METHOD exe : BOOL
VAR_INPUT
	emergency		:BOOL;		//signal of All_Block and Safety conditions
END_VAR
VAR_IN_OUT
	CMD				:udtCMD;	//standart command word
END_VAR
// Device mode determination
	IF NOT emergency THEN
		//Normal mode
		IF NOT CMD.force THEN
			//No technological lock
			IF NOT CMD.lock AND NOT CMD.alarm AND NOT CMD.service THEN
				//No manual mode
				IF NOT CMD.manual THEN
					CMD.startM := CMD.startA;
				END_IF;
			ELSE
				//Technological lock or device alarm
				CMD.startM := FALSE;
			END_IF;
		END_IF;
	ELSE
		//emergency stop
		CMD.startM := FALSE;
	END_IF;
END_METHOD

METHOD inc : INT
VAR_INPUT
	value			:INT;
	maxValue		:INT;
END_VAR
VAR_IN_OUT
	rotate			:BOOL;
END_VAR
IF rotate THEN
	inc := value + 1;
	IF inc > maxValue THEN
		inc := 0;
	END_IF
	rotate := FALSE;
ELSE
	inc := value;
END_IF
END_METHOD

METHOD blink : BOOL
VAR_INPUT
	req				:BOOL;
	clockOn			:timerRtc;
	clockOff		:timerRtc;
	spOn			:REAL;
	spOff			:REAL;
END_VAR
//blink method
IF req THEN
	//work time
	IF NOT clockOn.cmd.Q AND NOT clockOff.cmd.Q THEN
		blink := TRUE;
		clockOn.cmd.start := TRUE;
	END_IF
	//wait time
	IF clockOn.cmd.Q AND NOT clockOff.cmd.Q THEN
		blink := FALSE;
		clockOff.cmd.start := TRUE;
	END_IF
	//restart time
	IF clockOn.cmd.Q AND clockOff.cmd.Q THEN
		clockOn.cmd.start := FALSE;
		clockOFF.cmd.start := FALSE;
	END_IF
ELSE
	clockOn.cmd.start := FALSE;
	clockOFF.cmd.start := FALSE;
	blink := FALSE;
END_IF

clockOn.sp := spOn;
clockOff.sp := spOff;
sys.timer.rtc(clockOn);
sys.timer.rtc(clockOff);
END_METHOD

METHOD switch : BOOL
VAR_INPUT
	on				:BOOL;
	off				:BOOL;
END_VAR
IF NOT off AND on THEN
	switch := TRUE;
END_IF

IF off THEN
	switch := FALSE;
END_IF
END_METHOD

END_FUNCTION_BLOCK

// System/Library Methods/DrvTimer
FUNCTION_BLOCK DrvTimer
VAR_INPUT
END_VAR
VAR_OUTPUT
END_VAR
VAR
END_VAR

METHOD sec : BOOL
VAR_IN_OUT
	T			:timerSec;		//configuration and command struct for timer of seconds
END_VAR
// Timer with a multiplicity of 1 second
	IF T.CMD.start AND NOT T.CMD.reset THEN
		// Turn on
		IF T.ap < T.sp THEN
			IF NOT T.CMD.pause AND sys.pulse1s THEN
				T.ap := T.ap + 1;
			END_IF;
			T.CMD.Q := FALSE;
		ELSE
			// SP is achieved
			T.CMD.Q := TRUE;
		END_IF;
	ELSE
		// Turn off and reset
		T.ap := 0;
		T.CMD.Q := FALSE;
		T.CMD.reset := FALSE;
	END_IF;
END_METHOD

METHOD cnt : BOOL
VAR_INPUT
	signal 			:BOOL;			//signal from sensor or logical condition
END_VAR
VAR_IN_OUT
	T				:timerCnt;		//configuration and command struct for counter
END_VAR
// Front signal control
	T.PT (CLK := signal);
	
// Timer or counter with free multiplicity 
	IF T.CMD.start AND NOT T.CMD.reset THEN
		// Turn on
		IF NOT T.CMD.pause THEN
			IF T.PT.Q THEN
				T.ap := T.ap + T.one;
			END_IF;
		END_IF;
		//SP control
		IF T.ap < T.sp THEN
			// SP not achieved
			T.CMD.Q := FALSE;
		ELSE
			// SP is achieved
			T.CMD.Q := TRUE;
		END_IF;
	ELSE
		// Turn off and reset
		T.ap := 0.0;
		T.CMD.Q := FALSE;
		T.CMD.reset := FALSE;
	END_IF;

// Progress control
	IF T.sp > 0 AND T.CMD.start THEN
		IF T.ap <= T.sp THEN
			T.percent := (T.ap / T.sp) * 100.0;
		ELSE
			T.percent := 100;
		END_IF
	ELSE
		T.percent := 0.0;
	END_IF;
END_METHOD

METHOD rtc : BOOL
VAR_IN_OUT
	T			:timerRtc;			//configuration and command struct for timer of milliseconds
END_VAR
// Timer with a multiplicity of 1 second
		
	//time counting
	IF T.CMD.start AND NOT T.CMD.reset THEN
		// Turn on
			IF T.RTC = 0 THEN
				T.RTC := sys.upTimeMs;
			END_IF
		//delta calculate
			IF NOT T.CMD.Q THEN
				T.delta := sys.upTimeMs - T.RTC;
			END_IF;
		//delta control
		IF T.ap < T.sp THEN
			T.CMD.Q := FALSE;
		ELSE
			T.CMD.Q := TRUE;
		END_IF;
	ELSE
		// Turn off and reset
		T.ap := 0;
		T.RTC := 0;
		T.delta := 0;
		T.CMD.Q := FALSE;
		T.CMD.reset := FALSE;
	END_IF;
	
	//convert data
		T.ap := UDINT_TO_REAL(T.delta) / 1000;
	
	//calculate time
		IF T.sp > 0 AND T.CMD.start THEN
			T.percent := (T.ap / T.sp) * 100.0;
		ELSE
			T.percent := 0;
		END_IF;
END_METHOD

END_FUNCTION_BLOCK

// Drivers/Devices/03. Analog Input/DrvAI_MV210
FUNCTION_BLOCK DrvAI_MV210
VAR_INPUT
	signal			:udtAI_MV210_101;//Analog input signal from PLC
END_VAR	
VAR_IN_OUT
	CMD				:udtCMD;		//Non-retain structure with command word
	cfg				:cfgAI;			//Retain structure with settings
END_VAR
VAR_OUTPUT
	state			:stateAI_MV210;	//Non-retain structure with states information
	netData			:udtNetDataAnalog;	//Data for network communication via ModBus TCP/RTU
	result			:REAL;			//signal from sensor
END_VAR
VAR
	value			:REAL;			//tmp value for calculating 
	buffer			:REAL;			//tnp value for slow mode
	emergency		:BOOL;			//emergency signal
	cnt				:INT;			//internal counter
	PT				:ARRAY [0..1] OF R_TRIG;
	NT				:ARRAY [0..1] OF F_TRIG;
	clock			:ARRAY [0..3] OF timerRtc;
	Filter			:subFilter;
END_VAR

//ANALOG INPUT
//control of typical analog sensors
// - pressure
// - level
// - flowmeter
// - etc

s00_globalCommands();
IF NOT cfg.cfg.useCompact THEN
	//s01_externalCommand();
	s02_workMode();
	s03_filter();
	s04_alarmsRaw();
END_IF
s05_exe();
//s06_delays();
//s07_turnON();
//s08_turnOFF();
s09_options();
s10_alarms();
s11_reset();
s12_state();
//s13_commands();
//s14_opTime();
s15_globalData();
s16_timers();
s17_hmi();
s18_netData();
//s19_reserv();
//s20_test();

ACTION s07_turnON:

END_ACTION

ACTION s17_hmi:
//hmi data
	//input scaling
		state.signal := sys.base.scale(
			value := signal.signal,
			inputType := cfg.inputType,
			range := cfg.range);
	//rotate input type
		cfg.inputType := sys.base.inc(
			rotate := cmd.test,
			value := cfg.inputType,
			maxValue := sys.aiMaxValueType);
	//rotate value type
		cfg.valueType := sys.base.inc(
			rotate := cmd.lowSpeed,
			value := cfg.valueType,
			maxValue := sys.aiMaxValueValue);
	//rotate filter type
		cfg.filterType := sys.base.inc(
			rotate := cmd.local,
			value := cfg.filterType,
			maxValue := sys.aiMaxValueFilter);
END_ACTION

ACTION s04_alarmsRaw:
//alarms raw
	
	//SC control
	IF cfg.cfg.useSC AND CMD.startA  THEN
		CASE cfg.inputType OF 
			0: 	//0..20 mA
				state.alarm.almSC := sys.base.almS(
					signal := state.signal > 21.0,
					reset := cmd.reset);
			1: 	//4..20 mA
				state.alarm.almSC := sys.base.almS(
					signal := state.signal > 21.0,
					reset := cmd.reset);
				state.alarm.almNC := sys.base.almS(							//NC control only for 4..20 mA
					signal := state.signal < 2.5,
					reset := cmd.reset);
			2: 	//0..10 V
				state.alarm.almSC := sys.base.almS(
					signal := state.signal > 10.5,
					reset := cmd.reset);
			3: 	//-150..+150 C
				state.alarm.almSC := sys.base.almS(
					signal := state.signal > 155.0,
					reset := cmd.reset);
			4: 	//-150..+250 C
				state.alarm.almSC := sys.base.almS(
					signal := state.signal > 255.0,
					reset := cmd.reset);
			ELSE
				state.alarm.almSC := FALSE;
				state.alarm.almNC := FALSE;
		END_CASE
		//ST
		IF state.alarm.almNC OR state.alarm.almSC OR signal.errorCode > 0 THEN
			state.alarm.almST := TRUE;
		END_IF
		CASE signal.errorCode OF
			240:	state.alarm.INCORRECT_VALUE 		:= TRUE;
			241:	state.alarm.FIELDBUS_ERROR 			:= TRUE;
			246:	state.alarm.DATA_NOT_READY 			:= TRUE;
			247:	state.alarm.SENSOR_DISABLED 		:= TRUE;
			248:	state.alarm.TOO_HIGH_TEMP 			:= TRUE;
			249:	state.alarm.TOO_LOW_TEMP 			:= TRUE;
			250:	state.alarm.TOO_HIGH_VALUE 			:= TRUE;
			251:	state.alarm.TOO_LOW_VALUE 			:= TRUE;
			252:	state.alarm.SHORT_CIRCIUT 			:= TRUE;
			253:	state.alarm.SENSOR_FAILED 			:= TRUE;
			254:	state.alarm.NO_CONNECTION_TO_ADC 	:= TRUE;
			255:	state.alarm.INCORRECT_CALIBRATION 	:= TRUE;
		END_CASE
	ELSE
		state.alarm.almSC := FALSE;
		state.alarm.almNC := FALSE;
		state.alarm.almST := FALSE;
	end_if
END_ACTION

ACTION s00_globalCommands:
//global commands
	//emergency signal
		emergency := FALSE;
	//auto mode
		IF sys.allAuto THEN
			CMD.manual := FALSE;
		END_IF;
	//global reset
		IF sys.allreset THEN
			CMD.reset := TRUE;
		END_IF
END_ACTION

ACTION s10_alarms:
//alarms with time control
	//HH
		state.alarm.almHH := sys.base.alm(
			signal := (result > cfg.SP.HH AND cfg.cfg.useHigh),
			reset := (CMD.reset OR NOT CMD.startA) OR (cfg.cfg.useAutoReset AND result <= cfg.SP.HH),
			clock := clock[0].CMD);
	//H
		state.alarm.almH := sys.base.alm(
			signal := (result > cfg.SP.H),
			reset := (CMD.reset OR NOT CMD.startA OR (result < cfg.SP.H)),
			clock := clock[1].CMD);
	//L
		state.alarm.almL := sys.base.alm(
			signal := (result < cfg.SP.L),
			reset := (CMD.reset OR NOT CMD.startA OR (result > cfg.SP.L)),
			clock := clock[2].CMD);
	//LL
		state.alarm.almLL := sys.base.alm(
			signal := (result < cfg.SP.LL AND cfg.cfg.useLow),
			reset := (CMD.reset OR NOT CMD.startA) OR (cfg.cfg.useAutoReset AND result >= cfg.SP.LL),
			clock := clock[3].CMD);
END_ACTION

ACTION s11_reset:
//reset
	IF CMD.reset THEN
		state.state.alarm := FALSE;
		FOR cnt := 0 TO 3 DO
			clock[cnt].CMD.reset := TRUE;
		END_FOR
		state.alarm.INCORRECT_VALUE 		:= FALSE;
		state.alarm.FIELDBUS_ERROR 			:= FALSE;
		state.alarm.DATA_NOT_READY 			:= FALSE;
		state.alarm.SENSOR_DISABLED 		:= FALSE;
		state.alarm.TOO_HIGH_TEMP 			:= FALSE;
		state.alarm.TOO_LOW_TEMP 			:= FALSE;
		state.alarm.TOO_HIGH_VALUE 			:= FALSE;
		state.alarm.TOO_LOW_VALUE 			:= FALSE;
		state.alarm.SHORT_CIRCIUT 			:= FALSE;
		state.alarm.SENSOR_FAILED 			:= FALSE;
		state.alarm.NO_CONNECTION_TO_ADC 	:= FALSE;
		state.alarm.INCORRECT_CALIBRATION 	:= FALSE;
		CMD.alarm := FALSE;
		CMD.reset := FALSE;
	END_IF
END_ACTION

ACTION s16_timers:
//call timers
	FOR cnt := 0 TO 3 DO
		clock[cnt].SP := INT_TO_REAL(cfg.spT[cnt]) / 10.0;
		sys.timer.rtc (clock[cnt]);
	END_FOR
END_ACTION

ACTION s15_globalData:
//manual mode flag
	IF CMD.manual THEN sys.man.drvAI := TRUE; END_IF;
	
//global alarm
	IF (state.alarm.almST OR state.alarm.almHH OR state.alarm.almLL) AND CMD.startA THEN
		state.state.alarm := TRUE;
		sys.alm.drvAI := TRUE;
		CMD.alarm := TRUE;
	END_IF
END_ACTION

ACTION s02_workMode:
//convert data		
	cmd.startA := cfg.cfg.useEnable;
	//data convert to phisycal value scale
		value := sys.base.conv(
			signal := signal.signal,
			range := cfg.range);
			
	//signal's correction
		IF NOT CMD.startA THEN
			value := 0;
		ELSE
			value := value * cfg.Multiplier + cfg.Calibration;
		END_IF
END_ACTION

ACTION s03_filter:
//signal filter	
	//filtering mode
		Filter(
			start := CMD.startA AND cfg.cfg.useFilter,
			signal := value,
			filterType := cfg.filterType,
			filterLim := cfg.filterLim,
			result => buffer);
			
	//no filtering mode
		IF NOT cfg.cfg.useFilter THEN
			buffer := value;
		END_IF
END_ACTION

ACTION s05_exe:
//device control
	sys.base.exe(emergency := emergency,
		CMD := CMD);
END_ACTION

ACTION s06_delays:

END_ACTION

ACTION s08_turnOFF:

END_ACTION

ACTION s09_options:
//options
	IF cmd.startA THEN
		IF NOT cmd.manual THEN
			state.result := buffer;
		END_IF
	ELSE
		state.result := 0.0;
	END_IF
	
//state signal transfer	
	result := state.result;
END_ACTION

ACTION s12_state:
//state information
	cmd.call := TRUE;
END_ACTION

ACTION s18_netData:
netData.status 	:= state.status;
netData.ap 		:= state.result;
netData.alarm.0 := state.alarm.almST;
netData.alarm.1 := state.alarm.almHH;
//netData.alarm.2 := state.alarm.almH;
//netData.alarm.3 := state.alarm.almL;
netData.alarm.4 := state.alarm.almLL;
netData.alarm.5 := state.alarm.SENSOR_FAILED;
netData.alarm.6 := state.alarm.SHORT_CIRCIUT;
netData.alarm.7 := state.alarm.INCORRECT_VALUE;
netData.alarm.8 := state.alarm.TOO_HIGH_VALUE;
netData.alarm.9 := state.alarm.TOO_LOW_TEMP;
END_ACTION

END_FUNCTION_BLOCK

// Drivers/Devices/04. Analog Output/DrvAO_MV210
FUNCTION_Block DrvAO_MV210
VAR_INPUT
	command			:BOOL;			//Command in automation mode from algorythms
	setPoint		:REAL;			//Control signal from algorythm
END_VAR	
VAR_IN_OUT
	CMD				:udtCMD;		//Non-retain structure with command word
	cfg				:cfgAO;			//Retain structure with settings
	devState		:udtDevAnalog;	
	resultI			:udtAO_MV210_502;//Analog output signal to PLC in INT
END_VAR
VAR_OUTPUT
	state			:stateAO_MV210;	//Non-retain structure with states information
	netData			:udtNetDataAnalog;//Data for network communication via ModBus TCP/RTU
END_VAR
VAR
	value			:REAL;			//tmp value for calculating 
	buffer			:REAL;			//tnp value for slow mode
	emergency		:BOOL;			//emergency signal
	spA				:REAL;			//setpoint for work
	cnt				:INT;			//internal counter
	PT				:ARRAY [0..1] OF R_TRIG;
	NT				:ARRAY [0..1] OF F_TRIG;
	drvSlow			:subSlow;
END_VAR

//ANALOG OUTPUT
//control of typical analog command
// - Hz setpoint for motors
// - % setpoint for valves

s00_globalCommands();
s01_externalCommand();
//s02_workMode();
//s03_filter();
s04_alarmsRaw();
s05_exe();
//s06_delays();
//s07_turnON();
//s08_turnOFF();
s09_options();
//s10_alarms();
s11_reset();
s12_state();
//s13_commands();
//s14_opTime();
s15_globalData();
//s16_timers();
s17_hmi();
s18_netData();
//s19_reserv();
//s20_test();

ACTION s12_state:
//state information
	cmd.call := TRUE;
	//ready
		devState.READY := NOT cmd.lock AND NOT cmd.force AND NOT cmd.alarm AND NOT emergency;
	//busy
		devState.BUSY := cmd.startM AND cfg.spM <> buffer;
	//done
		devState.DONE := cmd.startM AND cfg.spM = buffer;
	//ap
		devState.AP := buffer;
END_ACTION

ACTION s17_hmi:
//hmi data
	//convert data
		state.signal := sys.base.scale(
			value := resultI.value,
			inputType := cfg.outputType,
			range := cfg.range);
	//rotate output type
		cfg.outputType := sys.base.inc(
			rotate := cmd.test,
			value := cfg.outputType,
			maxValue := sys.aoMaxValueType);
	//rotate value type
		cfg.valueType := sys.base.inc(
			rotate := cmd.lowSpeed,
			value := cfg.valueType,
			maxValue := sys.aoMaxValueValue);
	//HMI light
		IF cfg.cfg.useLight THEN
			IF CMD.startA THEN state.status := 1; END_IF
			IF NOT CMD.startA THEN state.status := 0; END_IF
		ELSE
			state.status := 0;
		END_IF
END_ACTION

ACTION s15_globalData:
//manual mode flag
	IF CMD.manual THEN sys.man.drvAO := TRUE; END_IF;
END_ACTION

ACTION s00_globalCommands:
//global commands
	//emergency signal
		IF cfg.cfg.useNoEmrg THEN
			emergency := FALSE;
		ELSE
			emergency := sys.allBlock;
		END_IF
	//to auto mode
		IF sys.allAuto THEN
			CMD.manual := FALSE;
		END_IF;
	//simulation mode
		PT[0](CLK := sys.allSim);
		NT[0](CLK := sys.allSim);
		IF PT[0].Q THEN cfg.cfg.useSim := TRUE; END_IF;
		IF NT[0].Q THEN cfg.cfg.useSim := FALSE; END_IF;
		IF cfg.cfg.useSim THEN sys.sim.drvAO := TRUE; END_IF;
END_ACTION

ACTION s01_externalCommand:
//select source of control
	IF cfg.cfg.useExt THEN
		CMD.startA := command;
		spA := setPoint;
	ELSE
		CMD.startA := devState.REQ;
		spA := devState.SP;
	END_IF
	IF NOT CMD.manual THEN
		cfg.spM := spA;
	END_IF
END_ACTION

ACTION s05_exe:
//device control
	sys.base.exe(emergency := emergency,
		CMD := CMD);
	//setpoint control
		IF NOT CMD.manual THEN
			cfg.spM := setPoint;
		END_IF
		IF NOT CMD.startM THEN
			cfg.spM := 0;
		END_IF
END_ACTION

ACTION s09_options:
//slow mode for analog output
	drvSlow(
		REQ := cfg.cfg.useSlow,
		signal := cfg.spM,
		cfg := cfg.slowCfg,
		state => state.slowState,
		result => buffer);

//data convert to phisycal value scale
	value := sys.base.conv(
		signal := buffer,
		range := cfg.range);
		
//state signal transfer
	state.result := buffer;
		
//simulation mode
	IF NOT cfg.cfg.useSim THEN
		resultI.value := REAL_TO_UINT(value);
	ELSE
		resultI.value := 0;
	END_IF
END_ACTION

ACTION s04_alarmsRaw:
//alarms raw
	
	//SC control
	IF CMD.startA  THEN
		IF resultI.errorCode > 0 THEN
			state.state.alarm := TRUE;
			CMD.alarm := true;
			sys.alm.drvAO := TRUE;
		END_IF
		CASE resultI.errorCode OF
			1:	state.almMV210.NO_DAC_CONNECTION 	:= TRUE;
			2:	state.almMV210.NO_LOAD 				:= TRUE;
			3:	state.almMV210.DAC_OVERHEAT 		:= TRUE;
			4:	state.almMV210.CRC_ERROR 			:= TRUE;
			5:	state.almMV210.CHANNEL_DISABLED 	:= TRUE;
			6:	state.almMV210.SHORT_CIRCUIT 		:= TRUE;
		END_CASE
	END_IF
END_ACTION

ACTION s11_reset:
//reset
	IF CMD.reset THEN
		state.state.alarm 					:= FALSE;
		state.almMV210.NO_DAC_CONNECTION 	:= FALSE;
		state.almMV210.NO_LOAD 				:= FALSE;
		state.almMV210.DAC_OVERHEAT 		:= FALSE;
		state.almMV210.CRC_ERROR 			:= FALSE;
		state.almMV210.CHANNEL_DISABLED 	:= FALSE;
		state.almMV210.SHORT_CIRCUIT 		:= FALSE;
		CMD.alarm := FALSE;
		CMD.reset := FALSE;
	END_IF
END_ACTION

ACTION s18_netData:
netData.status 	:= state.status;
netData.ap 		:= state.result;
netData.alarm.0 := state.almMV210.NO_LOAD;
netData.alarm.1 := state.almMV210.DAC_OVERHEAT;
netData.alarm.2 := state.almMV210.SHORT_CIRCUIT;
END_ACTION

END_FUNCTION_BLOCK

// System/Library UDTs/devAtoD
FUNCTION devAtoD : udtDevDiscrete
VAR_IN_OUT
	devA				:udtDevAnalog;
END_VAR
VAR
END_VAR

devAtoD.REQ := devA.REQ;

END_FUNCTION

// System/Library UDTs/devDtoA
FUNCTION devDtoA : udtDevAnalog
VAR_IN_OUT
	devD			:udtDevDiscrete;
END_VAR
VAR
END_VAR

devDtoA.REQ := devD.REQ;

END_FUNCTION

// Drivers/Special/DrvStatistics
FUNCTION_BLOCK DrvStatistics
VAR_INPUT
	enable			:BOOL;
	signalD			:BOOL;
	signalA			:REAL;
END_VAR
VAR_IN_OUT
	cfg				:cfgStatistic;
END_VAR
VAR_OUTPUT
END_VAR
VAR
	calcOk			:BOOL;
	multiplicator	:REAL := 1.0;
	value			:REAL;
	PT				:ARRAY [0..1] OF R_TRIG;
END_VAR

PT[0](CLK := signalD);

//calculate statistics
	IF cfg.useAnalog THEN
		cfg.useDiscrete := FALSE;
		IF NOT calcOk THEN
			calcMulti();
			calcOk := TRUE;
		END_IF
		IF cfg.useClock THEN
			calcA();
		ELSE
			IF sys.pulse01s THEN
				calcA();
			END_IF
		END_IF
	ELSE
		cfg.useDiscrete := TRUE;
	END_IF

ACTION calcD:
IF PT[0].Q THEN
	IF enable THEN
		cfg.work 	:= addValue(cfg.weightD, cfg.work);
		cfg.all		:= addValue(cfg.weightD, cfg.all);
	ELSE
		IF cfg.useSkip THEN
			cfg.skip	:= addValue(cfg.weightD, cfg.skip);
		END_IF
	END_IF
END_IF
END_ACTION

METHOD addValue : listStatistic
VAR_INPUT
	value			:REAL;
	list			:listStatistic;
END_VAR
addValue.seans 	:= list.seans + value;
addValue.hour 	:= list.hour + value;
addValue.day 	:= list.day + value;
addValue.week 	:= list.week + value;
addValue.month 	:= list.month + value;
addValue.year 	:= list.year + value;
addValue.total 	:= list.total + value;
END_METHOD

ACTION reset:
IF cfg.reset THEN
	cfg.resetWork 	:= TRUE;
	cfg.resetSkip 	:= TRUE;
	cfg.resetAll 	:= TRUE;
END_IF

IF cfg.resetWork THEN
	cfg.work := resetList(cfg.work);
	cfg.resetWork := FALSE;
END_IF

IF cfg.resetSkip THEN
	cfg.skip := resetList(cfg.skip);
	cfg.resetSkip := FALSE;
END_IF

IF cfg.resetAll THEN
	cfg.all := resetList(cfg.all);
	cfg.resetAll := FALSE;
END_IF
END_ACTION

METHOD resetList : listStatistic
VAR_IN_OUT
	list			:listStatistic;
END_VAR
resetList.hour 	:= 0.0;
resetList.day	:= 0.0;
resetList.week	:= 0.0;
resetList.month	:= 0.0;
resetList.year	:= 0.0;
resetList.total	:= 0.0;
END_METHOD

ACTION calcA:
value := signalA * multiplicator;
IF enable THEN
	cfg.work 	:= addValue(value, cfg.work);
	cfg.all		:= addValue(value, cfg.all);
ELSE
	IF cfg.useSkip THEN
		cfg.skip	:= addValue(value, cfg.skip);
	END_IF
END_IF
END_ACTION

ACTION calcMulti:
//calculate multiplicator
	IF NOT cfg.useClock THEN
		CASE cfg.weightA OF
			//0 - hour, 1 - minutes, 2 - seconds
			0:	multiplicator := 36000;
			1:	multiplicator := 600;
			2: 	multiplicator := 10;
		END_CASE
	ELSE
		CASE cfg.weightA OF
			//0 - hour, 1 - minutes, 2 - seconds
			0:	multiplicator := 3600 * (0.1 / cfg.weightClock);
			1:	multiplicator := 60 * (0.1 / cfg.weightClock);
			2: 	multiplicator := 1 * (0.1 / cfg.weightClock);
		END_CASE
	END_IF
END_ACTION

END_FUNCTION_BLOCK

// System/Library Methods/mbSwap
FUNCTION mbSwap : DWORD
VAR_INPUT
	source		:uniSwap;
END_VAR
VAR
	swapping	:uniSwap;
END_VAR

swapping.source[1] := source.source[0];
swapping.source[0] := source.source[1]; 
mbSwap := swapping.value;

END_FUNCTION

// System/DrvRetain
FUNCTION_BLOCK DrvRetain
VAR_INPUT
	retainFileName		:STRING;
END_VAR

VAR_OUTPUT
END_VAR
VAR
	step				:INT;						//step for process
	pApp				:POINTER TO APPLICATION;
	result              :RTS_IEC_RESULT; 			//Result code for operations
	fbDelete			:FILE.Delete; 				//Function block to delete the file
	//commands
	delete				:BOOL;
END_VAR

//works with retain memory
	fbDelete(
		xExecute := delete,
		xDone => ,
		xBusy => ,
		xError => ,
		sFileName := retainFileName,
		eError => );
		
system();

METHOD custom : BOOL
VAR_IN_OUT
	save				:BOOL;
	load				:BOOL;
END_VAR
//save to file
	IF save THEN
		CASE step OF
			0: //reset hmi connections
				sys.loadZero := TRUE;
				step := 1;
			1: //reset completed
				IF NOT sys.loadZero THEN
					step := 2;
				END_IF
			2: //delete file
				delete := TRUE;
				step := 3;
			3: //check delete
				IF fbDelete.xDone OR fbDelete.xError THEN
					delete := FALSE;
					IF NOT fbDelete.xBusy THEN
						step := 10;
					END_IF
				END_IF
			10: //save data to file
				pApp := AppGetCurrent(pResult:=ADR(Result));
				IF pApp <> 0 THEN
					(* Store the variables in a file*)
					Result := AppStoreRetainsInFile(pApp,retainFileName);
				END_IF
				step := 0;
				save := FALSE;
		END_CASE
	END_IF
	
//load from file
	IF load THEN
		CASE step OF
			0: //reset hmi connections
				sys.loadZero := TRUE;
				step := 1;
			1: //reset completed
				IF NOT sys.loadZero THEN
					step := 2;
				END_IF
			2:	//load data
				pApp := AppGetCurrent(pResult:=ADR(Result));
				Result := AppRestoreRetainsFromFile(pApp,retainFileName);
				load := FALSE;
				step := 0;
		END_CASE
	END_IF
END_METHOD

ACTION system:
//save to file
	IF sys.retainSave THEN
		CASE step OF
			0: //reset hmi connections
				sys.loadZero := TRUE;
				step := 1;
			1: //reset completed
				IF NOT sys.loadZero THEN
					step := 2;
				END_IF
			2: //delete file
				delete := TRUE;
				step := 3;
			3: //check delete
				IF fbDelete.xDone OR fbDelete.xError THEN
					delete := FALSE;
					IF NOT fbDelete.xBusy THEN
						step := 10;
					END_IF
				END_IF
			10: //save data to file
				pApp := AppGetCurrent(pResult:=ADR(Result));
				IF pApp <> 0 THEN
					(* Store the variables in a file*)
					Result := AppStoreRetainsInFile(pApp,retainFileName);
				END_IF
				step := 0;
				sys.retainSave := FALSE;
		END_CASE
	END_IF
	
//load from file
	IF sys.retainLoad THEN
		CASE step OF
			0: //reset hmi connections
				sys.loadZero := TRUE;
				step := 1;
			1: //reset completed
				IF NOT sys.loadZero THEN
					step := 2;
				END_IF
			2:	//load data
				pApp := AppGetCurrent(pResult:=ADR(Result));
				Result := AppRestoreRetainsFromFile(pApp,retainFileName);
				sys.retainLoad := FALSE;
				step := 0;
		END_CASE
	END_IF
END_ACTION

END_FUNCTION_BLOCK
